FUNCTION_BLOCK AdsConnector EXTENDS StateMachine
VAR_INPUT
END_VAR
VAR_OUTPUT
END_VAR
VAR
	fbStepWorkerBusy : FB_StepWorker;
	cbConnected : Boolean; //Custom Boolean
	fbAdsSupplier : AdsSupplier;
END_VAR

SUPER^();
Start();

METHOD PROTECTED Busy : BOOL
VAR_INPUT
END_VAR
VAR_INST
	eAdsConnectorBusy : E_AdsConnectorBusy;
END_VAR
eAdsConnectorBusy := fbStepWorkerBusy.getStep;
IF fbStepWorkerBusy.getStep = eNO_STEP 
THEN
	fbStepWorkerBusy.mNextStep(eCHECK_IF_CONNECTED);
END_IF


CASE fbStepWorkerBusy.getStep OF

	eCHECK_IF_CONNECTED:
	
		fbStepWorkerBusy.mAddCondition(cbConnected);
		fbStepWorkerBusy.mNextStep(eCONNECTED);
		
	eCONNECTED:
	
		fbAdsSupplier();
		IF NOT cbConnected.getValue
		THEN
			fbStepWorkerBusy.mNextStep(eDISCONNECTED);
		END_IF
	
	eDISCONNECTED:
	
		Done();
		fbStepWorkerBusy.mNextStep(eNO_STEP);
	
END_CASE
END_METHOD

METHOD PROTECTED  Error : BOOL
VAR_INPUT
END_VAR
END_METHOD

METHOD PROTECTED  Idle : BOOL
VAR_INPUT
END_VAR
END_METHOD

METHOD PROTECTED  Init : BOOL
VAR_INPUT
END_VAR
END_METHOD

METHOD PROTECTED  Prepare : BOOL
VAR_INPUT
END_VAR
END_METHOD

METHOD PROTECTED  Ready : BOOL
VAR_INPUT
END_VAR
END_METHOD

METHOD PROTECTED  Waiting : BOOL
VAR_INPUT
END_VAR
END_METHOD

END_FUNCTION_BLOCK

(* stored: Version 1.1.0.1, ProductVersion 3.1.4024.0
   POU AdsConnector: Id {d13dc3ab-3002-426d-a960-f2af687c2ce6}, SpecialFunc None
   Method Busy: Id {557bd86e-e555-4a7c-a77e-516b13eb9cf0}
   Method Error: Id {a1d17b9d-7981-4624-a63a-fd1f79acb21d}
   Method Idle: Id {49a1d8eb-b338-4a16-b4bf-a4091e30e9a6}
   Method Init: Id {dfdb3cd6-9bf2-430d-bc98-33debb6aea1b}
   Method Prepare: Id {ec94fc33-ef3b-440d-9e4e-8102bbd092c1}
   Method Ready: Id {97a24525-ce74-408c-8373-d4df1bf45d95}
   Method Waiting: Id {eae2389e-1940-4a75-9526-c10b28c969c3} *)
